(* IEC 61131-3 sources: stateaware-ics-monitoring/tests/st_gen/golden/ctown, 9 files *)

(* ---- ctown_plc1.st ---- *)
(* Auto-generated by st_gen from ctown.inp + ctown_plcs.yaml
   Topology: ctown   PLC: PLC1
   DO NOT EDIT. *)

PROGRAM PLC1
VAR_INPUT
    T1 : REAL;            (* sourced from PLC2 *)
END_VAR
VAR_OUTPUT
    PU1 : BOOL;
    PU2 : BOOL;
END_VAR
VAR
    PU1_State : INT := 0;
    PU2_State : INT := 0;
END_VAR

(* ----- FSM for actuator PU1 ----- *)
CASE PU1_State OF
    0:  (* CLOSED *)
        IF T1 < 4 THEN
            PU1_State := 1;
        END_IF;
    1:  (* OPEN *)
        IF T1 > 6.3 THEN
            PU1_State := 0;
        END_IF;
END_CASE;
PU1 := (PU1_State = 1);

(* ----- FSM for actuator PU2 ----- *)
CASE PU2_State OF
    0:  (* CLOSED *)
        IF T1 < 1 THEN
            PU2_State := 1;
        END_IF;
    1:  (* OPEN *)
        IF T1 > 4.5 THEN
            PU2_State := 0;
        END_IF;
END_CASE;
PU2 := (PU2_State = 1);

END_PROGRAM

(* ---- ctown_plc2.st ---- *)
(* Auto-generated by st_gen from ctown.inp + ctown_plcs.yaml
   Topology: ctown   PLC: PLC2
   DO NOT EDIT. *)

PROGRAM PLC2
(* No actuators with [CONTROLS] entries -- sensor-only or static-setting PLC. *)
END_PROGRAM

(* ---- ctown_plc3.st ---- *)
(* Auto-generated by st_gen from ctown.inp + ctown_plcs.yaml
   Topology: ctown   PLC: PLC3
   DO NOT EDIT. *)

PROGRAM PLC3
VAR_INPUT
    T2 : REAL;            (* owned by this PLC *)
    T3 : REAL;            (* sourced from PLC4 *)
    T4 : REAL;            (* sourced from PLC6 *)
END_VAR
VAR_OUTPUT
    V2 : BOOL;
    PU4 : BOOL;
    PU5 : BOOL;
    PU6 : BOOL;
    PU7 : BOOL;
END_VAR
VAR
    V2_State : INT := 0;
    PU4_State : INT := 0;
    PU5_State : INT := 0;
    PU6_State : INT := 0;
    PU7_State : INT := 0;
END_VAR

(* ----- FSM for actuator V2 ----- *)
CASE V2_State OF
    0:  (* CLOSED *)
        IF T2 < 0.5 THEN
            V2_State := 1;
        END_IF;
    1:  (* OPEN *)
        IF T2 > 5.5 THEN
            V2_State := 0;
        END_IF;
END_CASE;
V2 := (V2_State = 1);

(* ----- FSM for actuator PU4 ----- *)
CASE PU4_State OF
    0:  (* CLOSED *)
        IF T3 < 3 THEN
            PU4_State := 1;
        END_IF;
    1:  (* OPEN *)
        IF T3 > 5.3 THEN
            PU4_State := 0;
        END_IF;
END_CASE;
PU4 := (PU4_State = 1);

(* ----- FSM for actuator PU5 ----- *)
CASE PU5_State OF
    0:  (* CLOSED *)
        IF T3 < 1 THEN
            PU5_State := 1;
        END_IF;
    1:  (* OPEN *)
        IF T3 > 3.5 THEN
            PU5_State := 0;
        END_IF;
END_CASE;
PU5 := (PU5_State = 1);

(* ----- FSM for actuator PU6 ----- *)
CASE PU6_State OF
    0:  (* CLOSED *)
        IF T4 < 2 THEN
            PU6_State := 1;
        END_IF;
    1:  (* OPEN *)
        IF T4 > 3.5 THEN
            PU6_State := 0;
        END_IF;
END_CASE;
PU6 := (PU6_State = 1);

(* ----- FSM for actuator PU7 ----- *)
CASE PU7_State OF
    0:  (* CLOSED *)
        IF T4 < 3 THEN
            PU7_State := 1;
        END_IF;
    1:  (* OPEN *)
        IF T4 > 4.5 THEN
            PU7_State := 0;
        END_IF;
END_CASE;
PU7 := (PU7_State = 1);

END_PROGRAM

(* ---- ctown_plc4.st ---- *)
(* Auto-generated by st_gen from ctown.inp + ctown_plcs.yaml
   Topology: ctown   PLC: PLC4
   DO NOT EDIT. *)

PROGRAM PLC4
(* No actuators with [CONTROLS] entries -- sensor-only or static-setting PLC. *)
END_PROGRAM

(* ---- ctown_plc5.st ---- *)
(* Auto-generated by st_gen from ctown.inp + ctown_plcs.yaml
   Topology: ctown   PLC: PLC5
   DO NOT EDIT. *)

PROGRAM PLC5
VAR_INPUT
    T5 : REAL;            (* sourced from PLC7 *)
    T7 : REAL;            (* sourced from PLC9 *)
END_VAR
VAR_OUTPUT
    PU8 : BOOL;
    PU10 : BOOL;
    PU11 : BOOL;
END_VAR
VAR
    PU8_State : INT := 0;
    PU10_State : INT := 0;
    PU11_State : INT := 0;
END_VAR

(* ----- FSM for actuator PU8 ----- *)
CASE PU8_State OF
    0:  (* CLOSED *)
        IF T5 < 1.5 THEN
            PU8_State := 1;
        END_IF;
    1:  (* OPEN *)
        IF T5 > 4 THEN
            PU8_State := 0;
        END_IF;
END_CASE;
PU8 := (PU8_State = 1);

(* ----- FSM for actuator PU10 ----- *)
CASE PU10_State OF
    0:  (* CLOSED *)
        IF T7 < 1.5 THEN
            PU10_State := 1;
        END_IF;
    1:  (* OPEN *)
        IF T7 > 4.8 THEN
            PU10_State := 0;
        END_IF;
END_CASE;
PU10 := (PU10_State = 1);

(* ----- FSM for actuator PU11 ----- *)
CASE PU11_State OF
    0:  (* CLOSED *)
        IF T7 < 0.5 THEN
            PU11_State := 1;
        END_IF;
    1:  (* OPEN *)
        IF T7 > 3 THEN
            PU11_State := 0;
        END_IF;
END_CASE;
PU11 := (PU11_State = 1);

END_PROGRAM

(* ---- ctown_plc6.st ---- *)
(* Auto-generated by st_gen from ctown.inp + ctown_plcs.yaml
   Topology: ctown   PLC: PLC6
   DO NOT EDIT. *)

PROGRAM PLC6
(* No actuators with [CONTROLS] entries -- sensor-only or static-setting PLC. *)
END_PROGRAM

(* ---- ctown_plc7.st ---- *)
(* Auto-generated by st_gen from ctown.inp + ctown_plcs.yaml
   Topology: ctown   PLC: PLC7
   DO NOT EDIT. *)

PROGRAM PLC7
(* No actuators with [CONTROLS] entries -- sensor-only or static-setting PLC. *)
END_PROGRAM

(* ---- ctown_plc8.st ---- *)
(* Auto-generated by st_gen from ctown.inp + ctown_plcs.yaml
   Topology: ctown   PLC: PLC8
   DO NOT EDIT. *)

PROGRAM PLC8
(* No actuators with [CONTROLS] entries -- sensor-only or static-setting PLC. *)
END_PROGRAM

(* ---- ctown_plc9.st ---- *)
(* Auto-generated by st_gen from ctown.inp + ctown_plcs.yaml
   Topology: ctown   PLC: PLC9
   DO NOT EDIT. *)

PROGRAM PLC9
(* No actuators with [CONTROLS] entries -- sensor-only or static-setting PLC. *)
END_PROGRAM
